TYPE ST_ITC_Subsystem :
(**************************************************************************************
 * 	Application		:	BoxControl Framework
 *	Revision		:	$Revision: 404529 $
 *	Revision date	:	$Date: 2018-04-23 08:21:38 +0200 (Mo., 23 Apr 2018) $
 *	Last changed by	:	$Author: b7bolm $
 *	URL				:	$URL: http://almscdc.swisslog.com/repo/SWPD/Development/BoxControlFramework/20_Release/trunk/01_Software/BCF/BCF/JumpStart/20_Product/10_App/15_Subsystem/10_Lib/10_Conv/01_DUTs/ST_ITC_SubSystem.TcDUT $
 *
 *	Purpose			:	Subsystem ITC structure
 *
 * ------------------------------------------------------------------------------------
 *	Copyright Swisslog [IP AG], Switzerland. All rights reserved.
 * 
 * ------------------------------------------------------------------------------------
 *	
 * 	Revision History: 
 *
 * 	VERSION			DATE			INITIALS			DESCRIPTION
 *	0.1				01.01.2001		swl					Example
 *
 **************************************************************************************)
STRUCT
	Commands	: ST_ITC_SubsystemCommands; // Internal ITC commands
	Variable	: DINT; // Control variable
END_STRUCT
END_TYPE

(* stored: Version 1.1.0.1, ProductVersion 3.1.4022.12
   DUT ST_ITC_SubSystem: Id {f1914229-ed27-4236-b954-004c1bd3d0a3} *)
